(* PLC project tapis, TNI-Software ControlBuild 4.00 *)
(* stored: creationDateTime 2018-09-17T16:22:13-01:00 *)

CONFIGURATION tapis
  VAR_GLOBAL
    simuperiod : REAL := 50000.0;
    taskname : STRING(50) := 'tapis.exe';
    allowpreconditions : BOOL := true;
    allowpostconditions : BOOL := true;
  END_VAR
END_CONFIGURATION
